{attribute 'qualified_only'}
VAR_GLOBAL
	Error:  BOOL;
	Errors_Profinet_1:  WORD;
	Errors_Profinet_10:  Word;
	Errors_Profinet_11:  Word;
	Errors_Profinet_2:  Word;
	Errors_Profinet_3:  Word;
	Errors_Profinet_4:  Word;
	Errors_Profinet_5:  Word;
	Errors_Profinet_6:  Word;
	Errors_Profinet_7:  Word;
	Errors_Profinet_8:  Word;
	Errors_Profinet_9:  Word;
	Errors_Word_Gates_1:  Word;
	Errors_Word_Gates_2:  Word;
	Errors_Word_LightGuard_1:  Word;
	Errors_Word_Logistex:  Word;
	Errors_Word_Shuttles_1:  Word;
	Errors_Word_Shuttles_2:  Word;
	Erros_Supply_Feedback_1:  Word;
	Erros_Supply_Feedback_2:  Word;
	Erros_Supply_Feedback_3:  Word;
	Erros_Supply_Feedback_4:  Word;
	Erros_Supply_Feedback_5:  Word;
	Erros_Supply_Feedback_6:  Word;
	Erros_Supply_Feedback_7:  Word;
	Erros_Word_OPC_1:  Word;
	Erros_Word_OPC_2:  Word;
	Erros_Word_OPC_3:  Word;
	Erros_Word_OPC_4:  Word;
	Erros_Word_OPC_5:  Word;
	Estop_Error_Word_1:  Word;
	Estop_Error_Word_2:  Word;
	Estop_Error_Word_3:  Word;
	Estop_Error_Word_4:  Word;
	Estop_Error_Word_5:  Word;
	Estop_Error_Word_6:  Word;
	LE_Device_Errors_1:  WORD;
	LE_Device_Errors_2:  WORD;
	LE_Device_Errors_3:  WORD;
	LE_Device_Errors_4:  WORD;
	LE_Device_Errors_5:  WORD;
	LE_Warnings_1:  WORD;
	LE_Warnings_2:  WORD;
	LE_Warnings_3:  WORD;
	LE_Warnings_4:  WORD;
	LE_Warnings_5:  WORD;
	Barcode_Reader_ErrorCode_1:  WORD;
	Barcode_Reader_ErrorCode_1_2:  WORD;
	Barcode_Reader_ErrorCode_2:  WORD;
	Barcode_Reader_ErrorCode_2_2:  WORD;
	Barcode_Reader_ErrorCode_3:  WORD;
	Barcode_Reader_ErrorCode_3_2:  WORD;
	Barcode_Reader_ErrorCode_4:  WORD;
	Barcode_Reader_ErrorCode_4_2:  WORD;
	Barcode_Reader_ErrorCode_5:  WORD;
	Barcode_Reader_ErrorCode_5_2:  WORD;
END_VAR

(* stored: Version 1.1.0.1
   GVL Errors_GVL: Id {69f1f32d-7938-4835-af3d-cedf9cf8291a} *)
